FUNCTION_BLOCK StepperAxis EXTENDS ParentAxis
VAR
END_VAR

METHOD StartDisable : BOOL
StartDisable := TRUE;
RETURN;
END_METHOD

METHOD StartEnable : BOOL
StartEnable := TRUE;
RETURN;
END_METHOD

METHOD StartErrorChecking : BOOL
StartErrorChecking := TRUE;
RETURN;
END_METHOD

METHOD StartMovement : BOOL
StartMovement := TRUE;
RETURN;
END_METHOD

METHOD StartReset : BOOL
StartReset := TRUE;
RETURN;
END_METHOD

END_FUNCTION_BLOCK

(* stored: Version 1.1.0.1, ProductVersion 3.1.4024.12
   POU StepperAxis: Id {189fccae-bee1-415c-bc25-decf2c850847}, SpecialFunc None
   Folder METH: Id {1672590b-6e8e-48bd-903c-afc155b4d60c}
   Folder PROP: Id {abbce322-1fff-4209-8310-f27aff23493b}
   Method StartDisable: Id {9a766d63-1e7a-462b-bf96-77b749b909ea}
   Method StartEnable: Id {39dea5bd-28fb-4815-b413-9597368890df}
   Method StartErrorChecking: Id {76d84d50-a797-4ecc-a398-58ec3e382b6d}
   Method StartMovement: Id {d2cadbea-61fa-457c-b77f-e5833ab4054a}
   Method StartReset: Id {4a77efdd-6417-4e2a-bc4b-1cef098af65b} *)
